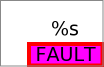
VISUALIZATION Obj_Healthy_Failed_Field  // 104x67
VAR_INPUT
	sIndex : STRING;
	bClosed : BOOL;
	bOffline : BOOL;
	bHealthy : BOOL;
END_VAR
    Rectangle (27,42 77x25), "%s", text list: 'CRAH_Isolator_Status', text index: bClosed
    Rectangle (27,16 76x26), "%s", text variable: sIndex
    Rectangle (27,42 77x25), "FAULT", invisible if: not bOffline
    Rectangle (27,42 77x25), invisible if: not bHealthy
END_VISUALIZATION

(* stored: Version 1.1.0.1, ProductVersion 3.1.4024.12
   Visu Obj_Healthy_Failed_Field: Id {f785296e-b220-4504-ad72-59cc7546bd0e} *)
